FUNCTION_BLOCK Reset (* Composite Function Block Type *)
  (* Standard: 61499-2 *)
  (* Version 0.0, 7/13/2026, Schneider Electric, template *)
  PACKAGE SE.Nereda;
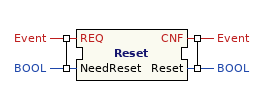
  EVENT_INPUT
    REQ WITH NeedReset; (* Normal Execution Request *)
  END_EVENT
  EVENT_OUTPUT
    CNF WITH Reset; (* Execution Confirmation *)
  END_EVENT
  VAR_INPUT
    NeedReset : BOOL;
  END_VAR
  VAR_OUTPUT
    Reset : BOOL;
  END_VAR
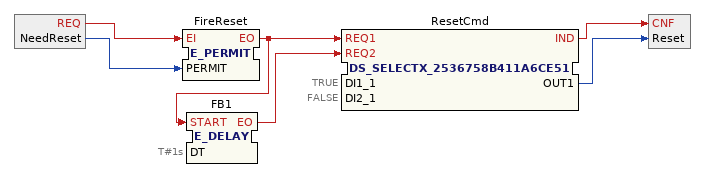
  FBS
    ResetCmd : DS_SELECTX_2536758B411A6CE51(DI1_1 := TRUE, DI2_1 := FALSE); {SET_ATTRIBUTE(Configuration.GenericFBType.InterfaceParams, Runtime.Standard#CNTX:=2;CNTY:=1;DI${CNTX,_,CNTY$}:BOOL)}
    FireReset : E_PERMIT;
    FB1 : E_DELAY(DT := T#1s);
  END_FBS
  EVENT_CONNECTIONS
    ResetCmd.IND TO CNF;
    FireReset.EO TO ResetCmd.REQ1;
    REQ TO FireReset.EI;
    FB1.EO TO ResetCmd.REQ2;
    FireReset.EO TO FB1.START;
  END_CONNECTIONS
  DATA_CONNECTIONS
    ResetCmd.OUT1 TO Reset;
    NeedReset TO FireReset.PERMIT;
  END_CONNECTIONS
END_FUNCTION_BLOCK
